TYPE Valve :
STRUCT
	bStart : BOOL;
	Output : BOOL;
	
	
END_STRUCT
END_TYPE

(* stored: Version 1.1.0.1, ProductVersion 3.1.4024.3
   DUT Valve: Id {beb88d00-84b7-461f-a91a-cdb473a3be38} *)
